FUNCTION_BLOCK UR5_StateMachine
VAR
//internal aux state
I_STATE : INT:=-1;
END_VAR


VAR_INPUT
	init_: BOOL:= FALSE;
	G_STATE: INT:=-1;
	Num_Ctr_Cam : INT:=-1;
END_VAR

VAR_OUTPUT
	State_complete : BOOL:= FALSE;
	Act_Gl_State :INT:=-1;
	Act_In_State: INT:=-1;
END_VAR

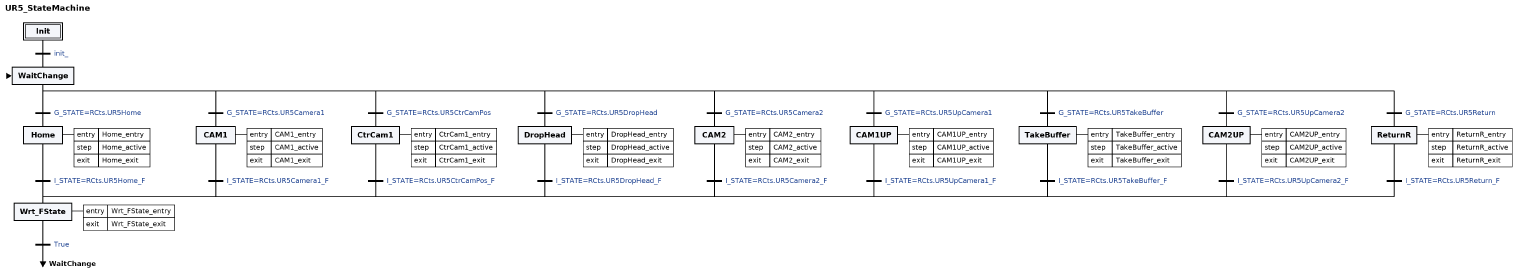
INITIAL_STEP Init:
END_STEP
TRANSITION FROM Init TO WaitChange
    := init_;
END_TRANSITION
STEP WaitChange:
END_STEP
TRANSITION FROM WaitChange TO Home
    := G_STATE=RCts.UR5Home;
END_TRANSITION
STEP Home:
    Home_entry(P1);  // entry action
    Home_active(N);  // step action
    Home_exit(P0);  // exit action
END_STEP
TRANSITION FROM Home TO Wrt_FState
    := I_STATE=RCts.UR5Home_F;
END_TRANSITION
TRANSITION FROM WaitChange TO CAM1
    := G_STATE=RCts.UR5Camera1;
END_TRANSITION
STEP CAM1:
    CAM1_entry(P1);  // entry action
    CAM1_active(N);  // step action
    CAM1_exit(P0);  // exit action
END_STEP
TRANSITION FROM CAM1 TO Wrt_FState
    := I_STATE=RCts.UR5Camera1_F;
END_TRANSITION
TRANSITION FROM WaitChange TO CtrCam1
    := G_STATE=RCts.UR5CtrCamPos;
END_TRANSITION
STEP CtrCam1:
    CtrCam1_entry(P1);  // entry action
    CtrCam1_active(N);  // step action
    CtrCam1_exit(P0);  // exit action
END_STEP
TRANSITION FROM CtrCam1 TO Wrt_FState
    := I_STATE=RCts.UR5CtrCamPos_F;
END_TRANSITION
TRANSITION FROM WaitChange TO DropHead
    := G_STATE=RCts.UR5DropHead;
END_TRANSITION
STEP DropHead:
    DropHead_entry(P1);  // entry action
    DropHead_active(N);  // step action
    DropHead_exit(P0);  // exit action
END_STEP
TRANSITION FROM DropHead TO Wrt_FState
    := I_STATE=RCts.UR5DropHead_F;
END_TRANSITION
TRANSITION FROM WaitChange TO CAM2
    := G_STATE=RCts.UR5Camera2;
END_TRANSITION
STEP CAM2:
    CAM2_entry(P1);  // entry action
    CAM2_active(N);  // step action
    CAM2_exit(P0);  // exit action
END_STEP
TRANSITION FROM CAM2 TO Wrt_FState
    := I_STATE=RCts.UR5Camera2_F;
END_TRANSITION
TRANSITION FROM WaitChange TO CAM1UP
    := G_STATE=RCts.UR5UpCamera1;
END_TRANSITION
STEP CAM1UP:
    CAM1UP_entry(P1);  // entry action
    CAM1UP_active(N);  // step action
    CAM1UP_exit(P0);  // exit action
END_STEP
TRANSITION FROM CAM1UP TO Wrt_FState
    := I_STATE=RCts.UR5UpCamera1_F;
END_TRANSITION
TRANSITION FROM WaitChange TO TakeBuffer
    := G_STATE=RCts.UR5TakeBuffer;
END_TRANSITION
STEP TakeBuffer:
    TakeBuffer_entry(P1);  // entry action
    TakeBuffer_active(N);  // step action
    TakeBuffer_exit(P0);  // exit action
END_STEP
TRANSITION FROM TakeBuffer TO Wrt_FState
    := I_STATE=RCts.UR5TakeBuffer_F;
END_TRANSITION
TRANSITION FROM WaitChange TO CAM2UP
    := G_STATE=RCts.UR5UpCamera2;
END_TRANSITION
STEP CAM2UP:
    CAM2UP_entry(P1);  // entry action
    CAM2UP_active(N);  // step action
    CAM2UP_exit(P0);  // exit action
END_STEP
TRANSITION FROM CAM2UP TO Wrt_FState
    := I_STATE=RCts.UR5UpCamera2_F;
END_TRANSITION
TRANSITION FROM WaitChange TO ReturnR
    := G_STATE=RCts.UR5Return;
END_TRANSITION
STEP ReturnR:
    ReturnR_entry(P1);  // entry action
    ReturnR_active(N);  // step action
    ReturnR_exit(P0);  // exit action
END_STEP
TRANSITION FROM ReturnR TO Wrt_FState
    := I_STATE=RCts.UR5Return_F;
END_TRANSITION
STEP Wrt_FState:
    Wrt_FState_entry(P1);  // entry action
    Wrt_FState_exit(P0);  // exit action
END_STEP
TRANSITION FROM Wrt_FState TO WaitChange
    := True;
END_TRANSITION

ACTION CAM1_active:
//read register from robot and chek is can read 2 or more correct values 
IF ck_state(RCts.UR5,RCts.UR5Camera1_I) THEN
	 I_STATE:= RCts.UR5Camera1_I;
ELSIF ck_state(RCts.UR5,RCts.UR5Camera1_F) THEN
	I_STATE := RCts.UR5Camera1_F;
END_IF

//read internal variable and write over output variable
Act_In_State := I_STATE;
END_ACTION

ACTION CAM1_entry:
//write state variables to robot, to execute respective state.
wr_state(RCts.UR5,RCts.UR5Camera1);
//write the retain state variable 
Act_Gl_State:=RCts.UR5Camera1;
END_ACTION

ACTION CAM1_exit:
//write reset state variables to robot.
wr_state(RCts.UR5,RCts.RESET_STATE);
//reset Global state variable
G_STATE := -1;
END_ACTION

ACTION CAM1UP_active:
//read register from robot and chek is can read 2 or more correct values 
IF ck_state(RCts.UR5,RCts.UR5UpCamera1_I) THEN
	 I_STATE:= RCts.UR5UpCamera1_I;
ELSIF ck_state(RCts.UR5,RCts.UR5UpCamera1_F) THEN
	I_STATE := RCts.UR5UpCamera1_F;
END_IF

//read internal variable and write over output variable
Act_In_State := I_STATE;
END_ACTION

ACTION CAM1UP_entry:
//write state variables to robot, to execute respective state.
wr_state(RCts.UR5,RCts.UR5UpCamera1);
//write the retain state variable 
Act_Gl_State:=RCts.UR5UpCamera1;
END_ACTION

ACTION CAM1UP_exit:
//write reset state variables to robot.
wr_state(RCts.UR5,RCts.RESET_STATE);
//reset Global state variable
G_STATE := -1;
END_ACTION

ACTION CAM2_active:
//read register from robot and chek is can read 2 or more correct values 
IF ck_state(RCts.UR5,RCts.UR5Camera2_I) THEN
	 I_STATE:= RCts.UR5Camera2_I;
ELSIF ck_state(RCts.UR5,RCts.UR5Camera2_F) THEN
	I_STATE := RCts.UR5Camera2_F;
END_IF



//read internal variable and write over output variable
Act_In_State := I_STATE;
END_ACTION

ACTION CAM2_entry:
//write state variables to robot, to execute respective state.
wr_state(RCts.UR5,RCts.UR5Camera2);
//write the retain state variable 
Act_Gl_State:=RCts.UR5Camera2;
END_ACTION

ACTION CAM2_exit:

//write reset state variables to robot.
wr_state(RCts.UR5,RCts.RESET_STATE);
//reset Global state variable
G_STATE := -1;
END_ACTION

ACTION CAM2UP_active:
//read register from robot and chek is can read 2 or more correct values 
IF ck_state(RCts.UR5,RCts.UR5UpCamera2_I) THEN
	 I_STATE:= RCts.UR5UpCamera2_I;
ELSIF ck_state(RCts.UR5,RCts.UR5UpCamera2_F) THEN
	I_STATE := RCts.UR5UpCamera2_F;
END_IF


//read internal variable and write over output variable
Act_In_State := I_STATE;
END_ACTION

ACTION CAM2UP_entry:
//write state variables to robot, to execute respective state.
wr_state(RCts.UR5,RCts.UR5UpCamera2);
//write the retain state variable 
Act_Gl_State:=RCts.UR5UpCamera2;
END_ACTION

ACTION CAM2UP_exit:
//write reset state variables to robot.
wr_state(RCts.UR5,RCts.RESET_STATE);
//reset Global state variable
G_STATE := -1;
END_ACTION

ACTION CtrCam1_active:

//read register from robot and chek is can read 2 or more correct values 
IF ck_state(RCts.UR5,RCts.UR5CtrCamPos_I) THEN
	 I_STATE:= RCts.UR5CtrCamPos_I;
ELSIF ck_state(RCts.UR5,RCts.UR5CtrCamPos_F) THEN
	I_STATE := RCts.UR5CtrCamPos_F;
END_IF


//read internal variable and write over output variable
Act_In_State := I_STATE;
END_ACTION

ACTION CtrCam1_entry:


CASE Num_Ctr_Cam OF 
	1:
		//write state variables to robot, to execute respective state.
		wr_state(RCts.UR5,RCts.UR5CtrCamPos1);
		//write the retain state variable 
		Act_Gl_State:=RCts.UR5CtrCamPos1;
	2:
		//write state variables to robot, to execute respective state.
		wr_state(RCts.UR5,RCts.UR5CtrCamPos2);
		//write the retain state variable 
		Act_Gl_State:=RCts.UR5CtrCamPos2;
	3:
		//write state variables to robot, to execute respective state.
		wr_state(RCts.UR5,RCts.UR5CtrCamPos3);
		//write the retain state variable 
		Act_Gl_State:=RCts.UR5CtrCamPos3;
	4:
		//write state variables to robot, to execute respective state.
		wr_state(RCts.UR5,RCts.UR5CtrCamPos4);
		//write the retain state variable 
		Act_Gl_State:=RCts.UR5CtrCamPos4;
	
END_CASE
END_ACTION

ACTION CtrCam1_exit:
//write reset state variables to robot.
wr_state(RCts.UR5,RCts.RESET_STATE);
//reset Global state variable
G_STATE := -1;
END_ACTION

ACTION DropHead_active:
//read register from robot and chek is can read 2 or more correct values 
IF ck_state(RCts.UR5,RCts.UR5DropHead_I) THEN
	 I_STATE:= RCts.UR5DropHead_I;
ELSIF ck_state(RCts.UR5,RCts.UR5DropHead_F) THEN
	I_STATE := RCts.UR5DropHead_F;
END_IF



//read internal variable and write over output variable
Act_In_State := I_STATE;
END_ACTION

ACTION DropHead_entry:
//write state variables to robot, to execute respective state.
wr_state(RCts.UR5,RCts.UR5DropHead);
//write the retain state variable 
Act_Gl_State:=RCts.UR5DropHead;
END_ACTION

ACTION DropHead_exit:

//write reset state variables to robot.
wr_state(RCts.UR5,RCts.RESET_STATE);
//reset Global state variable
G_STATE := -1;
END_ACTION

ACTION Home_active:
//read register from robot and chek is can read 2 or more correct values 
IF ck_state(RCts.UR5,RCts.UR5Home_I) THEN
	 I_STATE:= RCts.UR5Home_I;
ELSIF ck_state(RCts.UR5,RCts.UR5Home_F) THEN
	I_STATE := RCts.UR5Home_F;
END_IF


//read internal variable and write over output variable
Act_In_State := I_STATE;
END_ACTION

ACTION Home_entry:
//write state variables to robot, to execute respective state.
wr_state(RCts.UR5,RCts.UR5Home);
//write the retain state variable 
Act_Gl_State:=RCts.UR5Home;
END_ACTION

ACTION Home_exit:
//write reset state variables to robot.
wr_state(RCts.UR5,RCts.RESET_STATE);
//reset Global state variable
G_STATE := -1;
END_ACTION

ACTION ReturnR_active:
//read register from robot and chek is can read 2 or more correct values 
IF ck_state(RCts.UR5,RCts.UR5Return_I) THEN
	 I_STATE:= RCts.UR5Return_I;
ELSIF ck_state(RCts.UR5,RCts.UR5Return_F) THEN
	I_STATE := RCts.UR5Return_F;
END_IF


//read internal variable and write over output variable
Act_In_State := I_STATE;
END_ACTION

ACTION ReturnR_entry:
//write state variables to robot, to execute respective state.
wr_state(RCts.UR5,RCts.UR5Return);
//write the retain state variable 
Act_Gl_State:=RCts.UR5Return;
END_ACTION

ACTION ReturnR_exit:
//write reset state variables to robot.
wr_state(RCts.UR5,RCts.RESET_STATE);
//reset Global state variable
G_STATE := -1;
END_ACTION

ACTION TakeBuffer_active:
//read register from robot and chek is can read 2 or more correct values 
IF ck_state(RCts.UR5,RCts.UR5TakeBuffer_I) THEN
	 I_STATE:= RCts.UR5TakeBuffer_I;
ELSIF ck_state(RCts.UR5,RCts.UR5TakeBuffer_F) THEN
	I_STATE := RCts.UR5TakeBuffer_F;
END_IF

//read internal variable and write over output variable
Act_In_State := I_STATE;
END_ACTION

ACTION TakeBuffer_entry:
//write state variables to robot, to execute respective state.
wr_state(RCts.UR5,RCts.UR5TakeBuffer);
//write the retain state variable 
Act_Gl_State:=RCts.UR5TakeBuffer;
END_ACTION

ACTION TakeBuffer_exit:
//write reset state variables to robot.
wr_state(RCts.UR5,RCts.RESET_STATE);
//reset Global state variable
G_STATE := -1;
END_ACTION

ACTION Wrt_FState_entry:
//write output variable to indicate that the robot execute the state 
State_complete := TRUE;
END_ACTION

ACTION Wrt_FState_exit:
//write output variable to indicate that the robot execute the state 
State_complete := FALSE;
END_ACTION

END_FUNCTION_BLOCK

(* stored: Version 1.1.0.1, ProductVersion 3.1.4024.4
   POU UR5_StateMachine: Id {3400eb8f-1d25-4886-ac0c-ec707548dd2b}, SpecialFunc None
   Action CAM1_active: Id {5b26bb9e-700a-4e59-8d98-ba6ee4a380a7}
   Action CAM1_entry: Id {f5fe2ce2-ea1f-402b-9d4d-2af477ca2282}
   Action CAM1_exit: Id {00176d60-b24f-492d-85b5-a64e6ec86d80}
   Action CAM1UP_active: Id {e4620d80-7f6a-4c04-825b-6a6ad454dbcc}
   Action CAM1UP_entry: Id {2c045f69-4f07-404f-afa4-79983c55564c}
   Action CAM1UP_exit: Id {d588328e-aceb-4b04-873c-3c37bf40610d}
   Action CAM2_active: Id {5e52df75-004b-4656-b0d4-b12c00f56394}
   Action CAM2_entry: Id {100f546e-68bc-4ed7-9bbf-2f0f71186435}
   Action CAM2_exit: Id {b3f62bbf-86ed-4de1-8ce7-5e0405987826}
   Action CAM2UP_active: Id {f308dfca-c68f-4c41-b9a6-2c31f406ec8d}
   Action CAM2UP_entry: Id {bf932df4-1553-43cb-a7d4-eeef038c75ee}
   Action CAM2UP_exit: Id {98f6f2c1-0a65-4933-adbf-01798e116a99}
   Action CtrCam1_active: Id {5febf34f-b34e-4fc4-b5ee-9f9e3dc3915b}
   Action CtrCam1_entry: Id {75a959ed-4dea-4293-9ada-db11b5e0588f}
   Action CtrCam1_exit: Id {4bd831a3-45b0-4c58-a4bc-81a8ebf6d52e}
   Action DropHead_active: Id {d366534e-285c-4539-8591-4aac4301e9b0}
   Action DropHead_entry: Id {d6e9b0f0-74a9-45ee-b8ce-cadfbce390ff}
   Action DropHead_exit: Id {e41c4a84-e80b-4c0d-8064-ce4489343326}
   Action Home_active: Id {d39f8c31-9253-4419-b7d8-2b170ac80d66}
   Action Home_entry: Id {9ac03998-d4a7-407d-91af-4430256d0171}
   Action Home_exit: Id {00f3b8fc-4859-4352-a41c-094794dd05f3}
   Action ReturnR_active: Id {7556c092-86ce-41cb-952a-0afd53c61e4d}
   Action ReturnR_entry: Id {e9f51d88-4dd9-4ad7-aef2-0336d2ac78ac}
   Action ReturnR_exit: Id {ad89a8f6-6dc0-4abb-930e-216bfa91ab18}
   Action TakeBuffer_active: Id {23ce6aef-caa9-4f55-b03c-9c5bceb4c99e}
   Action TakeBuffer_entry: Id {c44c251c-37ba-4ec4-b21d-aa6b0fcb4de6}
   Action TakeBuffer_exit: Id {7f81b161-6305-4b2d-9a09-6cece059a1cb}
   Action Wrt_FState_entry: Id {9151d792-5d33-44de-b449-ede13ab3dcf3}
   Action Wrt_FState_exit: Id {3726172b-6a01-43f4-8c17-9c8dc3530286} *)
